// TIA Portal V17 export
// export: Created 2024-08-09T12:53:18.0421956Z, ExportSetting WithDefaults, DisplayName Totally Integrated Automation Portal, DisplayVersion V17 Update 7, DisplayName TIA Portal Openness, DisplayVersion V17 Update 7, DisplayName TIA Portal Version Control Interface, DisplayVersion V17, DisplayName STEP 7 Professional, DisplayVersion V17 Update 7, DisplayName STEP 7 Safety, DisplayVersion V17 Update 6, DisplayName WinCC Professional, DisplayVersion V17 Update 7
TYPE "S_ELT_TCEL"
// stored: IsFailsafeCompliant false
   STRUCT
      _Extrac { ExternalAccessible := 'False'; ExternalVisible := 'False'; ExternalWritable := 'False'} : Array[0.."NB_MOB_EXT"] of "S_CirExt";
      _Cel { ExternalAccessible := 'False'; ExternalVisible := 'False'; ExternalWritable := 'False'} : String["T_CD_CEL"];   // cellule d'extraction
      _Type { ExternalAccessible := 'False'; ExternalVisible := 'False'; ExternalWritable := 'False'} : USInt;   // Type cellule 1:origine 2:destination
      _NivHaut { ExternalAccessible := 'False'; ExternalVisible := 'False'; ExternalWritable := 'False'} : Bool;   // Niveau Haut
      _NivBas { ExternalAccessible := 'False'; ExternalVisible := 'False'; ExternalWritable := 'False'} : Bool;   // Niveau bas
      _NivInterm { ExternalAccessible := 'False'; ExternalVisible := 'False'; ExternalWritable := 'False'} : Bool;   // Niveau intermidiaire
      _Vibreur { ExternalAccessible := 'False'; ExternalVisible := 'False'; ExternalWritable := 'False'} : Bool;
   END_STRUCT;
END_TYPE
